# B&R Automation Studio project TestProject
Automation Studio 4.12.8.41 SP; technology packages: mappMotion 5.27.1

## Configuration X20CPU

CPU X20CP1686X, AutomationRuntime O4.93, Build 4.1.2, Vc V4.73.2

### Task classes (Cpu.sw)
```
Cyclic#1:
  Program <- Program.prg
Libraries: standard
```

### Hardware
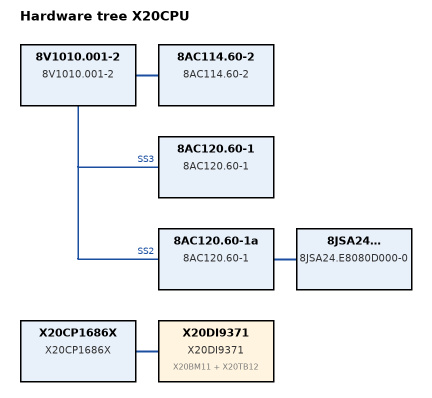
```
8AC114.60-2 : 8AC114.60-2 v1.0.0.8  [SS -> 8V1010.001-2.SS1; PLK1 -> X20CP1686X.IF3 (NodeNumber=1) [Cable Type=PowerlinkCable, Length=10, Version=1.0.0.3]]
8AC120.60-1 : 8AC120.60-1 v2.2.0.0  [SS -> 8V1010.001-2.SS3]
  PlugInType = Encoder
  McAcoposTypeID = AcoposPlugInConfig
8AC120.60-1a : 8AC120.60-1 v2.2.0.0  [SS -> 8V1010.001-2.SS2]
  PlugInType = Encoder
  McAcoposTypeID = AcoposPlugInConfig
8JSA24.E8080D000-0 : 8JSA24.E8080D000-0 v1.0.6.30  [EC -> 8AC120.60-1a.EC; MT -> 8V1010.001-2.MT1]
8V1010.001-2 : 8V1010.001-2 v2.2.0.0
  DriveConfiguration/Module:
    McAcoposTypeID = AcoposConfig
    ActivateACOPOSSimulationOnPLC = 0
  DriveConfiguration/Channel[1]/RealAxis:
    AxisReference = gAxis_1
    MechanicalElementsIsInvisible = 0
  DriveConfiguration/Channel[1]/RealAxis/MechanicalElements/Gearbox:
    InputIsReadOnly = 0
    Input = 1
    OutputIsReadOnly = 0
    Output = 1
  DriveConfiguration/Channel[1]/RealAxis/MechanicalElements/RotaryToLinearTransformation:
    ReferenceDistanceIsReadOnly = 0
    ReferenceDistance = 1
  DriveConfiguration/Channel[1]/RealAxis/Controller:
    ModeIsReadOnly = 0
    Mode = PositionController
  DriveConfiguration/Channel[1]/RealAxis/Controller/Mode/Position:
    ProportionalGain = 50.0
    IntegrationTime = 0.0
    PredictionTime = 0.0004
    TotalDelayTime = 0.0004
  DriveConfiguration/Channel[1]/RealAxis/Controller/Mode/Speed:
    ProportionalGainIsReadOnly = 0
    ProportionalGain = 2.0
    IntegrationTimeIsReadOnly = 0
    IntegrationTime = 0.0
    FilterTimeIsReadOnly = 0
    FilterTime = 0.0
  DriveConfiguration/Channel[1]/RealAxis/Controller/Mode/LoopFilters:
    LoopFilterXIsReadOnly = 0
    LoopFilter1 = NotUsed
    LoopFilter2 = NotUsed
    LoopFilter3 = NotUsed
  DriveConfiguration/Channel[1]/RealAxis/Homing:
    ModeIsReadOnly = 0
    Mode = Direct
  DriveConfiguration/Channel[1]/RealAxis/Homing/Mode:
    Position = 0.0
    ReferencePulse = NotUsed
  DriveConfiguration/Channel[1]/RealAxis/Homing:
    RestorePositionVariable = 
  DriveConfiguration/Channel[1]/RealAxis/StopReaction:
    QuickstopIsReadOnly = 0
    Quickstop = DecelerationLimit
    DriveErrorIsReadOnly = 0
    DriveError = DecelerationLimit
  DriveConfiguration/Channel[1]/RealAxis/MovementErrorLimits:
    PositionError = 1.0
    VelocityErrorMonitoring = Automatic1
  DriveConfiguration/Channel[1]/RealAxis:
    JerkFilterIsReadOnly = 0
    JerkFilter = NotUsed
    ZeroVibrationFilter = NotUsed
  DriveConfiguration/Channel[1]/RealAxis/DigitalInputs/HomingSwitch:
    SourceIsReadOnly = 0
    Source = X1Ref
    Level = High
  DriveConfiguration/Channel[1]/RealAxis/DigitalInputs/PositiveLimitSwitch:
    Source = X1PosLim
    Level = High
  DriveConfiguration/Channel[1]/RealAxis/DigitalInputs/NegativeLimitSwitch:
    Source = X1NegLim
    Level = High
  DriveConfiguration/Channel[1]/RealAxis/DigitalInputs/Trigger1:
    Source = X1Trigger1
    Level = High
  DriveConfiguration/Channel[1]/RealAxis/DigitalInputs/Trigger2:
    Source = X1Trigger2
    Level = High
  DriveConfiguration/Channel[1]/RealAxis/DigitalInputs/Quickstop:
    Input = Trigger2
  DriveConfiguration/Channel[1]/RealAxis/Simulation:
    SimulationModeOnPLC = SetValueGeneration
    SimulationModeOnACOPOS = NotUsed
  DriveConfiguration/Channel[1]:
    ExternalEncoderAxis = NotUsed
X20BM11 : X20BM11 v1.1.0.0  [X2X1 -> X20CP1686X.IF6]
X20CP1686X : X20CP1686X v1.6.2.0
  Connector IF2:
    ActivateDevice = 1
  ConfigurationID = TestProject_X20CPU
  Simulation = 1
  FileDevice1
  FileDeviceName1 = USER
  FileDevicePath1 = USER_PATH
  ActivateOpcUa = 1
  OpcUa_AuthenticationSecurityPolicy_EnableNone = 1
  OpcUa_AuthenticationSecurityPolicy_EnableBasic128Rsa15 = 1
  OpcUaInformationModels_PV_Version = 1
X20DI9371 : X20DI9371 v1.4.0.0  [SS1 -> X20TB12.SS; SL -> X20BM11.SL1]
X20TB12 : X20TB12 v1.0.0.0
```

### TestAxes.axis - X20CP1686X/mappMotion/TestAxes.axis
```
Element gAxis_1 (Type=axis)
  BaseTypeIsReadOnly = 0
  BaseType = LinearBounded
    MeasurementUnit = 5066068
    MeasurementResolutionIsReadOnly = 0
    MeasurementResolution = 0.01
    CountDirectionIsReadOnly = 0
    CountDirection = Standard
  MovementLimitsIsReadOnly = 0
  MovementLimits = Internal
    Position:
      LowerLimitMin = -1.79769313486231E308
      UpperLimitMax = 1.79769313486231E308
      LowerLimit = -1000.0
      UpperLimit = 1000.0
    VelocityIsReadOnly = 0
    Velocity:
      VelocityMax = 3.4E38
      Velocity = 50.0
    AccelerationIsReadOnly = 0
    Acceleration:
      AccelerationMax = 3.4E38
      Acceleration = 50.0
    DecelerationIsReadOnly = 0
    Deceleration:
      DecelerationMax = 3.4E38
      Deceleration = 50.0
  Alarms = None
```

## Logical view

Binary libraries used (declarations not repeated): operator, runtime, astime, AsIecCon, standard, MpAxis 5.27.1, McAxis 5.27.1, MpBase, McBase 5.27.1, McAcpAx 5.27.1, csvfilelib, fiowrap, hmitools, logthat, piper, ringbuflib, stringext, FileIO, sys_lib, AsBrStr, AsArLog, AsBrWStr, ArEventLog

### Global.var - Global variables
```iecst
VAR
	gMachine : Piper_typ;
END_VAR
```

### Package Logical/Libraries - Global libraries

### IO.typ
```iecst
TYPE
	IO_Pusher_typ : 	STRUCT
		aoActualPosition : REAL;
		diPusherExtended : BOOL;
		diPusherRetracted : BOOL;
		doPusherExtend : BOOL;
		doPusherRetract : BOOL;
	END_STRUCT;
	IO_typ : 	STRUCT
		conveyor : ARRAY[0..MAI_CONVEYORS]OF IO_Conveyor_typ;
		spawnCase : BOOL;
		pusher : IO_Pusher_typ;
	END_STRUCT;
	IO_Conveyor_typ : 	STRUCT
		diPhotoeyeEntrance : BOOL;
		diPhotoeyeExit : BOOL;
		doRunForward : BOOL;
		doRunReverse : BOOL;
		aoRunSpeed : REAL;
	END_STRUCT;
END_TYPE
```

### IO.var
```iecst
VAR
	io : IO_typ;
END_VAR
VAR CONSTANT
	MAX_CONVEYORS : UDINT := 4;
	MAI_CONVEYORS : UDINT := MAX_CONVEYORS-1;
END_VAR
```

### Program Logical/motionProgram (IEC)

#### Main.st - Init, cyclic, exit code
```iecst
PROGRAM _INIT

END_PROGRAM

PROGRAM _CYCLIC

	PiperModuleInterface;

	conveyor[3].downstreamReadyToReceive := TRUE;

	MapInputs;

	///// Timer Init

	counter := counter +1;

	FOR convIdx := 0 TO MAI_CONVEYORS DO
		conveyor[convIdx].overrun();
	END_FOR

	/////////Axis Handler

	IF NOT axisInit THEN

		IF NOT axisHandler.Active THEN
			axisHandler.Enable := TRUE;

		ELSIF NOT axisHandler.PowerOn THEN
			axisHandler.Power := TRUE;

		ELSIF NOT axisHandler.IsHomed THEN
			axisHandler.Home := TRUE;

		ELSE

			axisInit := TRUE;

		END_IF

		axisHandler.MpLink := ADR(gAxis_1);
		axisHandler.Parameters := ADR(axisParameters);

	ELSE

		io.pusher.aoActualPosition := 100 * LREAL_TO_REAL(axisHandler.Position);

		//// Case Logic

		FOR convIdx := 0 TO MAI_CONVEYORS DO

			CASE conveyor[convIdx].state OF

				WAITING_FOR_PACKAGE:

					conveyor[convIdx].runForward := FALSE;
					conveyor[convIdx].readyToReceive := TRUE;

					IF conveyor[convIdx].startOfConveyor THEN
						conveyor[convIdx].readyToReceive := FALSE;
						conveyor[convIdx].runForward := TRUE;

						conveyor[convIdx].state := HAS_PACKAGE;
					END_IF

				HAS_PACKAGE:

					conveyor[convIdx].readyToReceive := FALSE;

					IF NOT conveyor[convIdx].endOfConveyor AND NOT pushResetFlag THEN
						conveyor[convIdx].runForward := TRUE;

					ELSIF conveyor[convIdx].endOfConveyor THEN
						conveyor[convIdx].state := READY_TO_SEND_PACKAGE;

					ELSIF pushResetFlag THEN
						conveyor[2].state := WAITING_FOR_PACKAGE;
						pushResetFlag := FALSE;

					ELSE conveyor[convIdx].runForward := FALSE;

					END_IF

				READY_TO_SEND_PACKAGE:

					conveyor[convIdx].runForward := FALSE;

					IF conveyor[convIdx].downstreamReadyToReceive THEN
						conveyor[convIdx].state := SENDING_PACKAGE;

					END_IF

				SENDING_PACKAGE:

					conveyor[convIdx].runForward := TRUE;

					IF NOT conveyor[convIdx].downstreamReadyToReceive THEN
						conveyor[convIdx].state := WAITING_FOR_PACKAGE;

					ELSIF conveyor[3].endOfConveyor_ AND NOT conveyor[3].endOfConveyor THEN
						conveyor[3].state := WAITING_FOR_PACKAGE;
					END_IF

			END_CASE

		END_FOR

		IF gMachine.OUT.State =  MACH_ST_STARTING THEN
			io.spawnCase := TRUE;
		END_IF

		IF NOT conveyor[0].readyToReceive THEN
			io.spawnCase := FALSE;
		END_IF

		/////////// Spawner logic
		IF NOT conveyor[0].readyToReceive THEN
			spawnTimer.IN := TRUE;
		END_IF

		IF spawnTimer.Q AND conveyor[0].readyToReceive THEN
			io.spawnCase := TRUE;
			spawnTimer.IN := FALSE;
		END_IF

		//////// Case Length Logic

		IF conveyor[2].startOfConveyor THEN
			caseLengthTimer.IN := TRUE;
		END_IF

		IF conveyor[2].startOfConveyor_ AND NOT conveyor[2].startOfConveyor THEN
			caseLength := caseLengthTimer.ET;
			caseLengthTimer.IN := FALSE;
		END_IF

		///// Pusher Logic ////

		CASE pusherState OF

			WAITING:
				io.pusher.doPusherRetract := FALSE;
				IF caseLength >= T#600ms THEN
					pusherState := EXTENDING;
				END_IF

			EXTENDING:
				io.pusher.doPusherExtend := TRUE;
				IF io.pusher.diPusherExtended THEN
					io.pusher.doPusherExtend := FALSE;
					pusherState := EXTENDED;
				END_IF

			EXTENDED:
				axisHandler.MoveAbsolute := FALSE;
				IF NOT axisHandler.MoveAbsolute AND io.pusher.diPusherExtended THEN
					caseLength := T#0ms;
					pushResetFlag := TRUE;
					pusherState := RETRACTING;
				END_IF

			RETRACTING:
				io.pusher.doPusherRetract := TRUE;
				IF io.pusher.diPusherRetracted THEN
					io.pusher.doPusherRetract := FALSE;
					pusherState := RETRACTED;
				END_IF

			RETRACTED:
				axisHandler.MoveAbsolute := FALSE;
				IF NOT axisHandler.MoveAbsolute AND io.pusher.diPusherRetracted THEN
					pusherState := WAITING;
				END_IF

		END_CASE

	END_IF
	//////// Last scan for falling edge
	FOR convIdx := 0 TO MAI_CONVEYORS DO
		conveyor[convIdx].endOfConveyor_ := conveyor[convIdx].endOfConveyor;
		conveyor[convIdx].startOfConveyor_ := conveyor[convIdx].startOfConveyor;
	END_FOR

	///// Call Functions /////

	axisHandler();
	spawnTimer();
	pushReset();
	caseLengthTimer();

	MapOutputs;

END_PROGRAM

PROGRAM _EXIT

END_PROGRAM
```

#### Types.typ - Local data types
```iecst
TYPE
	State_enum :
		(
		WAITING_FOR_PACKAGE,
		HAS_PACKAGE,
		READY_TO_SEND_PACKAGE,
		RECEIVING_PACKAGE,
		SENDING_PACKAGE
		);
	Conveyor_type : 	STRUCT
		conveyorBusy : BOOL;
		startOfConveyor_ : BOOL;
		startOfConveyor : BOOL;
		endOfConveyor_ : BOOL;
		endOfConveyor : BOOL;
		overrun : TON := (PT:=T#750ms);
		runForward : BOOL;
		runRerverse : BOOL;
		readyToReceive : BOOL;
		readyToSend : BOOL;
		upstreamReadyToSend : BOOL;
		downstreamReadyToReceive : BOOL;
		state : State_enum;
	END_STRUCT;
	PusherState_enum :
		(
		WAITING,
		EXTENDING,
		RETRACTING,
		RETRACTED,
		EXTENDED
		);
END_TYPE
```

#### Variables.var - Local variables
```iecst
VAR
	spawnTimer : TON := (PT:=T#4000ms);
	pushReset : TON := (PT:=T#2000ms);
	counter : UDINT;
	convIdx : UDINT;
	conveyor : ARRAY[0..MAI_CONVEYORS] OF Conveyor_type;
	caseLengthTimer : TON := (PT:=T#10000ms);
	caseLength : TIME;
	axisParameters : MpAxisBasicParType;
	axisHandler : MpAxisBasic;
	axisInit : BOOL;
	systemTimer : TON;
	pusherState : PusherState_enum;
	pushResetFlag : BOOL;
	startFlag : BOOL;
END_VAR
```

#### MapOutputs.st
```iecst
ACTION MapOutputs:

	FOR convIdx := 0 TO MAI_CONVEYORS DO
		io.conveyor[convIdx].doRunForward := conveyor[convIdx].runForward AND startFlag;
		io.conveyor[convIdx].doRunReverse := conveyor[convIdx].runRerverse;
	END_FOR

	IF io.pusher.aoActualPosition = 500 THEN
		io.pusher.diPusherExtended := TRUE;
		io.pusher.diPusherRetracted := FALSE;
	END_IF

	IF io.pusher.aoActualPosition = 0 THEN
		io.pusher.diPusherRetracted := TRUE;
		io.pusher.diPusherExtended := FALSE;
	END_IF

	IF io.pusher.doPusherExtend THEN
		axisParameters.Position := 5;
		axisHandler.MoveAbsolute := TRUE;
	END_IF

	IF io.pusher.doPusherRetract THEN
		axisParameters.Position := 0;
		axisHandler.MoveAbsolute := TRUE;
	END_IF

END_ACTION
```

#### PiperModuleInterface.st
```iecst
// PiperModuleInterface.st
ACTION PiperModuleInterface:

	//Give this module a name so it is easier to debug
	ModuleInterface.ModuleName:=	'programUsingPiper';

	//Add a module to the Piper
	Module.ModuleInterface:=	ADR(ModuleInterface);
	Module.Piper:= 	ADR(gMachine);
	Module();

	// Handle any machine states that this module needs to respond to
	CASE ModuleInterface.PiperState OF
		//MACH_ST_BOOTING:
		//MACH_ST_CLEARING
		//MACH_ST_STOPPED:

		MACH_ST_STARTING:
			startFlag := TRUE;
			ModuleInterface.ModuleResponse:=	ModuleInterface.PiperState;

		//MACH_ST_IDLE:
		//MACH_ST_SUSPENDED:
		MACH_ST_EXECUTE:
			startFlag := TRUE;
		//MACH_ST_STOPPING:
		//		MACH_ST_ABORTING:
		//		MACH_ST_ABORTED:
		//		MACH_ST_HOLDING:
		//		MACH_ST_HELD:
		//		MACH_ST_UNHOLDING:
		//		MACH_ST_SUSPENDING:
		//		MACH_ST_UNSUSPENDING:
		//		MACH_ST_RESETTING:
		//		MACH_ST_COMPLETING:
		//		MACH_ST_COMPLETE:

		MACH_ST_BYPASSED:

		ELSE
			ModuleInterface.ModuleResponse:=	ModuleInterface.PiperState;
			startFlag := FALSE;
	END_CASE

END_ACTION
```

### Program Logical/Sequencing/Logic (IEC)

#### Main.st - Init, cyclic, exit code
```iecst
PROGRAM _INIT

	FOR index := 0 TO MAI_CONVEYORS DO
		conveyor[index].in.beltSpeed := 1.4;
	END_FOR

	processTimer.PT := T#1.7s;

	io;

END_PROGRAM

PROGRAM _CYCLIC

	MapInputs;

	// Map conveyor outputs to neighboring conveyor inputs.
	conveyor[0].in.downstreamReadyToReceive := conveyor[1].out.readyToReceive;
	conveyor[0].in.upstreamReadyToSend := TRUE;
	conveyor[1].in.downstreamReadyToReceive := conveyor[2].out.readyToReceive;
	conveyor[1].in.upstreamReadyToSend := conveyor[0].out.readyToSend;
	conveyor[2].in.downstreamReadyToReceive := conveyor[3].out.readyToReceive;
	conveyor[2].in.upstreamReadyToSend := conveyor[1].out.readyToSend;
	conveyor[3].in.downstreamReadyToReceive := conveyor[4].out.readyToReceive;
	conveyor[3].in.upstreamReadyToSend := conveyor[2].out.readyToSend;
	conveyor[4].in.downstreamReadyToReceive := processTimer.Q;
	conveyor[4].in.upstreamReadyToSend := conveyor[3].out.readyToSend;

	FOR index := 0 TO MAI_CONVEYORS DO

		// Reset all output signal cyclically.
		conveyor[index].out.readyToReceive := FALSE;
		conveyor[index].out.readyToSend := FALSE;
		conveyor[index].out.transferComplete := FALSE;
		conveyor[index].io.doRunForward := FALSE;

		CASE conveyor[index].internal.state OF

			CONVEYOR_ST_INIT:
				IF (conveyor[index].io.diPhotoeye2) THEN
					conveyor[index].internal.state := CONVEYOR_ST_READY_TO_SEND;
				ELSE
					conveyor[index].internal.state := CONVEYOR_ST_READY_TO_RECEIVE;
				END_IF

			CONVEYOR_ST_READY_TO_RECEIVE:
				conveyor[index].out.readyToReceive := TRUE;
				IF (conveyor[index].io.diPhotoeye1) THEN
					conveyor[index].internal.state := CONVEYOR_ST_RECEIVING;
				END_IF

			CONVEYOR_ST_RECEIVING:
				conveyor[index].out.readyToReceive := TRUE;
				conveyor[index].io.doRunForward := TRUE;
				IF (NOT conveyor[index].io.diPhotoeye1) THEN
					conveyor[index].internal.state := CONVEYOR_ST_POSITION;
				END_IF

			CONVEYOR_ST_POSITION:
				conveyor[index].io.doRunForward := TRUE;;
				IF (conveyor[index].io.diPhotoeye2) THEN
					IF (conveyor[index].in.downstreamReadyToReceive) THEN
						conveyor[index].internal.state := CONVEYOR_ST_SENDING;
					ELSE
						conveyor[index].internal.state := CONVEYOR_ST_READY_TO_SEND;
					END_IF
				END_IF

			CONVEYOR_ST_READY_TO_SEND:
				conveyor[index].out.readyToSend := TRUE;
				IF (conveyor[index].in.downstreamReadyToReceive) THEN
					conveyor[index].internal.state := CONVEYOR_ST_SENDING;
				END_IF

			CONVEYOR_ST_SENDING:
				conveyor[index].out.readyToSend := TRUE;
				conveyor[index].io.doRunForward := TRUE;
				IF (NOT conveyor[index].io.diPhotoeye2) THEN
					conveyor[index].internal.state := CONVEYOR_ST_READY_TO_RECEIVE;
				END_IF

		END_CASE

	END_FOR

	// Handle process logic.
	processTimer.IN := conveyor[4].out.readyToSend;
	processTimer();
	processActive := processTimer.IN;

	MapOutputs;

END_PROGRAM
```

#### Types.typ - Local data types
```iecst
TYPE
	Conveyor_Io_typ : 	STRUCT
		diPhotoeye1 : BOOL;
		diPhotoeye2 : BOOL;
		doRunForward : BOOL;
		doRunReverse : BOOL;
	END_STRUCT;
	Conveyor_Out_typ : 	STRUCT
		readyToSend : BOOL;
		readyToReceive : BOOL;
		transferComplete : BOOL;
	END_STRUCT;
	Conveyor_In_typ : 	STRUCT
		upstreamReadyToSend : BOOL;
		downstreamReadyToReceive : BOOL;
		beltSpeed : REAL;
	END_STRUCT;
	Conveyor_Internal_typ : 	STRUCT
		state : CONVEYOR_ST_enum;
	END_STRUCT;
	CONVEYOR_ST_enum :
		(
		CONVEYOR_ST_INIT,
		CONVEYOR_ST_READY_TO_RECEIVE,
		CONVEYOR_ST_RECEIVING,
		CONVEYOR_ST_POSITION,
		CONVEYOR_ST_READY_TO_SEND,
		CONVEYOR_ST_SENDING
		);
	Conveyor_typ : 	STRUCT
		in : Conveyor_In_typ;
		out : Conveyor_Out_typ;
		io : Conveyor_Io_typ;
		internal : Conveyor_Internal_typ;
	END_STRUCT;
END_TYPE
```

#### Variables.var - Local variables
```iecst
VAR
	conveyor : ARRAY[0..MAI_CONVEYORS] OF Conveyor_typ;
END_VAR
VAR CONSTANT
	MAI_CONVEYORS : USINT := 4;
END_VAR
VAR
	processTimer : TON;
	index : USINT;
	processActive : BOOL;
END_VAR
```

#### MapInputs.st
```iecst
ACTION MapInputs:

	FOR index := 0 TO MAI_CONVEYORS DO
		conveyor[index].io.diPhotoeye1 := io.conveyor[index].diPhotoeyeEntrance;
		conveyor[index].io.diPhotoeye2 := io.conveyor[index].diPhotoeyeExit;
	END_FOR

END_ACTION
```

#### MapOutputs.st
```iecst
ACTION MapOutputs:

	FOR index := 0 TO MAI_CONVEYORS DO
		io.conveyor[index].doRunForward := conveyor[index].io.doRunForward;
		io.conveyor[index].doRunReverse := conveyor[index].io.doRunReverse;
	END_FOR

END_ACTION
```

### Program Logical/piperProgram (IEC)

#### Main.st
```iecst
PROGRAM _INIT
	(* Insert code here *)

END_PROGRAM

PROGRAM _CYCLIC

	Piper_fn_Cyclic(gMachine);

END_PROGRAM

PROGRAM _EXIT
	(* Insert code here *)

END_PROGRAM
```

### Program Logical/programUsingPiper (IEC)

#### Main.st - Init, cyclic, exit code
```iecst
PROGRAM _INIT

END_PROGRAM

PROGRAM _CYCLIC

	PiperModuleInterface;

END_PROGRAM

PROGRAM _EXIT

END_PROGRAM
```

#### Types.typ - Local data types
```iecst
TYPE
	State_enum :
		(
		ST_IDLE,
		ST_RUNNING,
		New_Member1
		);
END_TYPE
```

#### Variables.var - Local variables
```iecst
VAR
	counter : UDINT;
	piperState : State_enum;
END_VAR
```

#### PiperModuleInterfaceTemplate.var
```iecst
VAR

	ModuleInterface : Module_Interface_typ;
	Module : Piper_Module_Fub;

END_VAR

VAR CONSTANT

END_VAR
```

#### PiperModuleInterface.st
```iecst
// PiperModuleInterface.st
ACTION PiperModuleInterface:

	//Give this module a name so it is easier to debug
	ModuleInterface.ModuleName:=	'programUsingPiper';

	//Add a module to the Piper
	Module.ModuleInterface:=	ADR(ModuleInterface);
	Module.Piper:= 	ADR(gMachine);
	Module();

	// Handle any machine states that this module needs to respond to
	CASE ModuleInterface.PiperState OF
		//		MACH_ST_BOOTING:
		//		MACH_ST_CLEARING:
		//		MACH_ST_STOPPED:
		//		MACH_ST_STARTING:
		//		MACH_ST_IDLE:
		//		MACH_ST_SUSPENDED:
		//		MACH_ST_EXECUTE:
		//		MACH_ST_STOPPING:
		//		MACH_ST_ABORTING:
		//		MACH_ST_ABORTED:
		//		MACH_ST_HOLDING:
		//		MACH_ST_HELD:
		//		MACH_ST_UNHOLDING:
		//		MACH_ST_SUSPENDING:
		//		MACH_ST_UNSUSPENDING:
		MACH_ST_RESETTING:
			counter := counter + 1 ;
			IF counter >= 400 THEN
				ModuleInterface.ModuleResponse:=	ModuleInterface.PiperState;
			END_IF
		//		MACH_ST_COMPLETING:
		//		MACH_ST_COMPLETE:

		MACH_ST_BYPASSED:

		ELSE
			ModuleInterface.ModuleResponse:=	ModuleInterface.PiperState;

	END_CASE

END_ACTION
```

#### MapInputs.st - not listed in the package file held
```iecst
ACTION MapInputs:

	FOR convIdx := 0 TO MAI_CONVEYORS DO
		conveyor[convIdx].startOfConveyor := io.conveyor[convIdx].diPhotoeyeEntrance;
		conveyor[convIdx].endOfConveyor := io.conveyor[convIdx].diPhotoeyeExit;
	END_FOR

	conveyor[0].downstreamReadyToReceive := conveyor[1].readyToReceive;

	conveyor[1].downstreamReadyToReceive := conveyor[2].readyToReceive;
	conveyor[1].upstreamReadyToSend:= conveyor[0].readyToSend;

	conveyor[2].downstreamReadyToReceive := conveyor[3].readyToReceive;
	conveyor[2].upstreamReadyToSend := conveyor[1].readyToSend;

	conveyor[3].upstreamReadyToSend := conveyor[0].readyToSend;

END_ACTION
```

#### MapOutputs.st - not listed in the package file held
```iecst
ACTION MapOutputs:

	FOR convIdx := 0 TO MAI_CONVEYORS DO
		io.conveyor[convIdx].doRunForward := conveyor[convIdx].runForward;
		io.conveyor[convIdx].doRunReverse := conveyor[convIdx].runRerverse;
	END_FOR

	IF io.pusher.aoActualPosition = 500 THEN
		io.pusher.diPusherExtended := TRUE;
		io.pusher.diPusherRetracted := FALSE;
	END_IF

	IF io.pusher.aoActualPosition = 0 THEN
		io.pusher.diPusherRetracted := TRUE;
		io.pusher.diPusherExtended := FALSE;
	END_IF

	IF io.pusher.doPusherExtend THEN
		axisParameters.Position := 5;
		axisHandler.MoveAbsolute := TRUE;
	END_IF

	IF io.pusher.doPusherRetract THEN
		axisParameters.Position := 0;
		axisHandler.MoveAbsolute := TRUE;
	END_IF

END_ACTION
```

### Program Logical/Program

#### Types.typ
```iecst
TYPE
	State_enum :
		(
		WAITING_FOR_PACKAGE,
		HAS_PACKAGE,
		READY_TO_SEND_PACKAGE,
		RECIEVING_PACKAGE,
		SENDING_PACKAGE
		);
	Task_typ : 	STRUCT
		status : Task_Status_typ;
	END_STRUCT;
	Task_Status_typ : 	STRUCT
		zone : ARRAY[0..MAI_CONVEYORS]OF Zone_type;
	END_STRUCT;
	Zone_type : 	STRUCT
		zoneBusy : BOOL;
		startOfZone_ : BOOL;
		startOfZone : BOOL;
		endOfZone_ : BOOL;
		endOfZone : BOOL;
		overrun : TON := (PT:=T#500ms);
		runForward : BOOL;
		runRerverse : BOOL;
		readyToReceive : BOOL;
		readyToSend : BOOL;
		upstreamReadyToSend : BOOL;
		downstreamReadyToReceive : BOOL;
		state : State_enum;
	END_STRUCT;
END_TYPE
```

#### Variables.var
```iecst
VAR
	convIdx : UDINT;
	counter : UDINT;
	spawnReset : TON := (PT:=T#1000ms);
	spawnTimer : TON := (PT:=T#4000ms);
	task : Task_typ;
	axis1Handler : MpAxisBasic;
	axis1Parameters : MpAxisBasicParType;
END_VAR
```

#### Main.st
```iecst
PROGRAM _INIT

END_PROGRAM

PROGRAM _CYCLIC

	MapInputs;

	///// Timer Init
	counter := counter +1;
	spawnTimer();
	spawnReset();
	FOR convIdx := 0 TO MAI_CONVEYORS DO
		task.status.zone[convIdx].overrun();
	END_FOR

	axis1Handler.MpLink := ADR(gAxis_1);
	axis1Handler.Parameters := ADR(axis1Parameters);
	axis1Handler.Enable := TRUE;

	io.pusher.aoActualPosition := 100 * LREAL_TO_REAL(axis1Handler.Position);

//////// Case Logic

	FOR convIdx := 0 TO MAI_CONVEYORS DO

		CASE task.status.zone[convIdx].state OF

			WAITING_FOR_PACKAGE:

				task.status.zone[convIdx].runForward := FALSE;
				task.status.zone[convIdx].readyToReceive := TRUE;

				IF task.status.zone[convIdx].startOfZone THEN
					task.status.zone[convIdx].readyToReceive := FALSE;
					task.status.zone[convIdx].runForward := TRUE;

					task.status.zone[convIdx].state := HAS_PACKAGE;
				END_IF

			HAS_PACKAGE:

				task.status.zone[convIdx].runForward := TRUE;

				IF task.status.zone[convIdx].endOfZone AND NOT task.status.zone[convIdx].downstreamReadyToReceive THEN
					task.status.zone[convIdx].state := READY_TO_SEND_PACKAGE;

				ELSIF task.status.zone[convIdx].endOfZone AND task.status.zone[convIdx].downstreamReadyToReceive THEN
					task.status.zone[convIdx].state:= SENDING_PACKAGE;
				END_IF

			READY_TO_SEND_PACKAGE:
				task.status.zone[convIdx].runForward := FALSE;
				IF task.status.zone[convIdx].downstreamReadyToReceive THEN
					task.status.zone[convIdx].state := SENDING_PACKAGE;
				END_IF

			SENDING_PACKAGE:
				task.status.zone[convIdx].runForward := TRUE;
				IF NOT task.status.zone[convIdx].endOfZone
				AND task.status.zone[convIdx].endOfZone_
				AND NOT task.status.zone[convIdx].downstreamReadyToReceive THEN
					task.status.zone[convIdx].state := WAITING_FOR_PACKAGE;
				END_IF

		END_CASE

	END_FOR

//////// Zone Busy State Logic
	FOR convIdx := 0 TO MAI_CONVEYORS DO
		IF task.status.zone[convIdx].startOfZone THEN
			task.status.zone[convIdx].zoneBusy := TRUE;
		ELSIF task.status.zone[convIdx].endOfZone_ AND NOT task.status.zone[convIdx].endOfZone THEN
			task.status.zone[convIdx].zoneBusy := FALSE;
		END_IF
	END_FOR

/////////// Spawner logic
	IF task.status.zone[0].zoneBusy THEN
		spawnTimer.IN := TRUE;
	END_IF

	IF spawnTimer.Q THEN
		io.spawnCase := TRUE;
		spawnTimer.IN := FALSE;
	END_IF

//////////// Conveyor Run Logic
	FOR convIdx := 0 TO MAI_CONVEYORS DO
		IF task.status.zone[convIdx].zoneBusy OR task.status.zone[convIdx].overrun.IN AND NOT task.status.zone[convIdx].overrun.Q THEN
			io.conveyor[convIdx].doRunForward := TRUE;
		ELSE
			io.conveyor[convIdx].doRunForward := FALSE;
		END_IF
	END_FOR

/////////// Overrun timer Logic
	FOR convIdx := 0 TO MAI_CONVEYORS DO
		IF NOT task.status.zone[convIdx].endOfZone AND task.status.zone[convIdx].endOfZone_ THEN
			task.status.zone[convIdx].overrun.IN := TRUE;
		END_IF
	END_FOR

	FOR convIdx := 0 TO MAI_CONVEYORS DO
		IF task.status.zone[convIdx].overrun.Q THEN
			task.status.zone[convIdx].overrun.IN:= FALSE;
		END_IF
	END_FOR
//
//////// Last scan for falling edge
		FOR convIdx := 0 TO MAI_CONVEYORS DO
		task.status.zone[convIdx].endOfZone_ := task.status.zone[convIdx].endOfZone;
		END_FOR

	MapOutputs;
	axis1Handler();

END_PROGRAM

PROGRAM _EXIT

END_PROGRAM
```

#### MapInputs.st
```iecst
ACTION MapInputs:

	FOR convIdx := 0 TO MAI_CONVEYORS DO
		task.status.zone[convIdx].startOfZone := io.conveyor[convIdx].diPhotoeyeEntrance;
		task.status.zone[convIdx].endOfZone := io.conveyor[convIdx].diPhotoeyeExit;
	END_FOR

	task.status.zone[0].downstreamReadyToReceive := task.status.zone[1].readyToReceive;

	task.status.zone[1].downstreamReadyToReceive := task.status.zone[2].readyToReceive;
	task.status.zone[1].upstreamReadyToSend:= task.status.zone[0].readyToSend;

	task.status.zone[2].downstreamReadyToReceive := task.status.zone[3].readyToReceive;
	task.status.zone[2].upstreamReadyToSend := task.status.zone[1].readyToSend;

	task.status.zone[3].upstreamReadyToSend := task.status.zone[0].readyToSend;

END_ACTION
```

#### MapOutputs.st
```iecst
ACTION MapOutputs:

	FOR convIdx := 0 TO MAI_CONVEYORS DO
		io.conveyor[convIdx].doRunForward := task.status.zone[convIdx].runForward;
		io.conveyor[convIdx].doRunReverse := task.status.zone[convIdx].runRerverse;
	END_FOR

END_ACTION
```

Listed in the project but not available here: Logical/Global.typ, Logical/motionProgram/MapInputs.st, Logical/motionProgram/PiperModuleInterfaceTemplate.var
